TYPE ST_Parameters_PCR :
STRUCT
	CalibrationNo		: INT;
    userID             	: STRING;
    density	            : STRING;
    solventNo           : STRING;
    solventRevision	    : STRING;
    allowableFail		: STRING;
    replicates	        : STRING;
    callInterval	    : STRING;
	sysRevisionNo		: INT;
END_STRUCT
END_TYPE

(* stored: Version 1.1.0.1, ProductVersion 3.1.4024.15
   DUT ST_Parameters_PCR: Id {95040081-31c9-44c3-9662-dee4256ad368} *)
